SUBAPPLICATION mapping_Uebung_010b5 (* SoftKey_F1-8 auf DigitalOutput_Q1-8 *)
  (* Standard: 61499-2; Description: Copyright (c) 2023 Meisterschulen am Ostbahnhof This program and the accompanying materials are made available under the terms of the Eclipse Public License 2.0 which is available at https://www.eclipse.org/legal/epl-2.0/ SPDX-License-Identifier: EPL-2.0 *)
  (* Version 1.0, 2023-10-23, Franz Höpfinger, Meisterschulen am Ostbahnhof *)
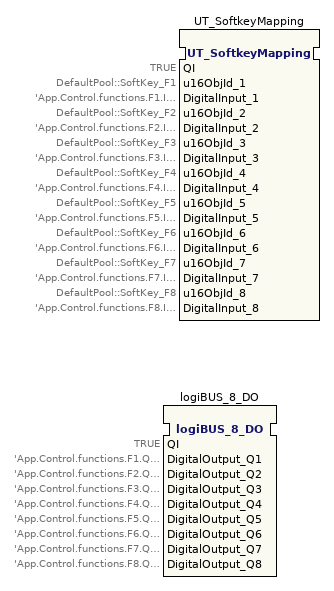
  FBS
    logiBUS_8_DO : logiBUS_8_DO(QI := TRUE, DigitalOutput_Q1 := 'App.Control.functions.F1.QX', DigitalOutput_Q2 := 'App.Control.functions.F2.QX', DigitalOutput_Q3 := 'App.Control.functions.F3.QX', DigitalOutput_Q4 := 'App.Control.functions.F4.QX', DigitalOutput_Q5 := 'App.Control.functions.F5.QX', DigitalOutput_Q6 := 'App.Control.functions.F6.QX', DigitalOutput_Q7 := 'App.Control.functions.F7.QX', DigitalOutput_Q8 := 'App.Control.functions.F8.QX');
    UT_SoftkeyMapping : UT_SoftkeyMapping(QI := TRUE, u16ObjId_1 := DefaultPool::SoftKey_F1, DigitalInput_1 := 'App.Control.functions.F1.IX', u16ObjId_2 := DefaultPool::SoftKey_F2, DigitalInput_2 := 'App.Control.functions.F2.IX', u16ObjId_3 := DefaultPool::SoftKey_F3, DigitalInput_3 := 'App.Control.functions.F3.IX', u16ObjId_4 := DefaultPool::SoftKey_F4, DigitalInput_4 := 'App.Control.functions.F4.IX', u16ObjId_5 := DefaultPool::SoftKey_F5, DigitalInput_5 := 'App.Control.functions.F5.IX', u16ObjId_6 := DefaultPool::SoftKey_F6, DigitalInput_6 := 'App.Control.functions.F6.IX', u16ObjId_7 := DefaultPool::SoftKey_F7, DigitalInput_7 := 'App.Control.functions.F7.IX', u16ObjId_8 := DefaultPool::SoftKey_F8, DigitalInput_8 := 'App.Control.functions.F8.IX');
  END_FBS
END_SUBAPPLICATION
